Fanuc KAREL source: kt00971.KL

-- PROVISIONAL review KL for V940-1; original PC SHA256 e9b38668dd76d0eae43348cff5972561d50aa5700ddd431d7c0e4aadaad1acdd
-- Incomplete behavior may be omitted. Consult companion uncertainty JSON. Do not deploy.
PROGRAM KT00971
%NOLOCKGROUP
BEGIN
  -- V9_ZERO_TABLE_METADATA_HINT layout=0001; no indexed target words; source/name/runtime held
  -- UNRESOLVED_PC offsets 5-12; opcodes 9C,23
  -- UNRESOLVED_PC offsets 17-25; opcodes 3F,75
  -- UNRESOLVED_PC offsets 30-43; opcodes 3F,75
  -- UNRESOLVED_PC offsets 48-86; opcodes 27,22,22,2A,22,2A,22,22,B0
  -- UNRESOLVED_PC offsets 91-95; opcodes 7F
END KT00971
